// TIA Portal V16 export
// export: Created 2021-09-01T08:19:45.4683166Z, ExportSetting WithDefaults, DisplayName Totally Integrated Automation Portal, DisplayVersion V16 Update 3, DisplayName TIA Portal Version Control Interface, DisplayVersion V16 Update 2, DisplayName TIA Portal Openness, DisplayVersion V16 Update 3, DisplayName TIA Portal Teamcenter Gateway, DisplayVersion V16, DisplayName STEP 7 Professional, DisplayVersion V16 Update 3, DisplayName STEP 7 Safety, DisplayVersion V16, DisplayName WinCC Advanced, DisplayVersion V16 Update 3
VAR_GLOBAL   // PLC tag table "CONST"
END_VAR
VAR_GLOBAL CONSTANT   // user constants
   MAX_STEP_NUMB : Int := 50;
   MIN_STEP_NUMB : Int := 1;
   MAX_DEV_NUMB : Int := 16;
   MIN_DEV_NUMB : Int := 1;
END_VAR
